FUNCTION_BLOCK CROSSCOMM_SENDER_2468F13B453622E42 (* Service Interface Function Block Type *)
  (* Standard: 61499-2 *)
  (* Version 0.0, 9/22/2017, bababen, nxtControl GmbH, template *)
  PACKAGE Main;
  (* Compiler Cpp nxtControl builtin 1.0 *)
  {SET_ATTRIBUTE(Runtime.FBType.ImplementingType, Runtime.System#DYNGEN_CROSSCOMM_SENDER)}
  {SET_ATTRIBUTE(Configuration.GenericFBType.InterfaceParams, Runtime.System#<InterfaceList> <EventInputs> <Event Name="CNF"> <With Var="PRetracked" /> <With Var="PExtended" /> </Event> </EventInputs> <InputVars> <VarDeclaration Name="PRetracked" Type="BOOL" /> <VarDeclaration Name="PExtended" Type="BOOL" /> </InputVars> </InterfaceList>)}
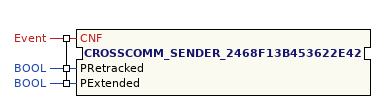
  EVENT_INPUT
    CNF WITH PRetracked, PExtended;
  END_EVENT
  VAR_INPUT
    PRetracked : BOOL;
    PExtended : BOOL;
  END_VAR
  EC_STATES
    START;
  END_STATES
END_FUNCTION_BLOCK
